// TIA Portal V19 export
FUNCTION "Conv_DT_to_STRING" : String   // FC39, LAD
// stored: Access Published, SetENOAutomatically false
   VAR_INPUT
      Val : DTL;
   END_VAR
   VAR_TEMP
      s_Y : String;
      s_M : String;
      s_D : String;
      s_H : String;
      s_Mi : String;
      s_S : String;
      s_N : String;
      str : String;
   END_VAR
BEGIN

REGION Network 1 (SCL)
   #s_Y := UINT_TO_STRING(#Val.YEAR);
   // Elimina il + a inizio stringa
   #s_Y := MID_STRING(IN := #s_Y, L := LEN(#s_Y) - 1, P := 2);



   #s_M := USINT_TO_STRING(#Val.MONTH);
   // Elimina il + a inizio stringa
   #s_M := MID_STRING(IN := #s_M, L := LEN(#s_M) - 1, P := 2);
   // Aggiunge lo 0 davanti per i mesi da 1 a 9
   IF LEN(#s_M) < 2 THEN
       #s_M := CONCAT(IN1 := '0', IN2 := #s_M);
   END_IF;



   #s_D := USINT_TO_STRING(#Val.DAY);
   // Elimina il + a inizio stringa
   #s_D := MID_STRING(IN := #s_D, L := LEN(#s_D) - 1, P := 2);
   // Aggiunge lo 0 davanti per i giorni da 1 a 9
   IF LEN(#s_D) < 2 THEN
       #s_D := CONCAT(IN1 := '0', IN2 := #s_D);
   END_IF;


   #s_H := USINT_TO_STRING(#Val.HOUR);
   // Elimina il + a inizio stringa
   #s_H := MID_STRING(IN := #s_H, L := LEN(#s_H) - 1, P := 2);
   // Aggiunge lo 0 davanti per le ore da 0 a 9
   IF LEN(#s_H) < 2 THEN
       #s_H := CONCAT(IN1 := '0', IN2 := #s_H);
   END_IF;


   #s_Mi := USINT_TO_STRING(#Val.MINUTE);
   // Elimina il + a inizio stringa
   #s_Mi := MID_STRING(IN := #s_Mi, L := LEN(#s_Mi) - 1, P := 2);
   // Aggiunge lo 0 davanti per i minuti da 0 a 9
   IF LEN(#s_Mi) < 2 THEN
       #s_Mi := CONCAT(IN1 := '0', IN2 := #s_Mi);
   END_IF;



   #s_S := USINT_TO_STRING(#Val.SECOND);
   // Elimina il + a inizio stringa
   #s_S := MID_STRING(IN := #s_S, L := LEN(#s_S) - 1, P := 2);
   // Aggiunge lo 0 davanti per i secondi da 0 a 9
   IF LEN(#s_S) < 2 THEN
       #s_S := CONCAT(IN1 := '0', IN2 := #s_S);
   END_IF;


   #s_N := UDINT_TO_STRING(#Val.NANOSECOND);
   // Elimina il + a inizio stringa
   #s_N := MID_STRING(IN := #s_N, L := LEN(#s_N) - 1, P := 2);
   // Riduci la string a solo 3 caratteri
   #s_N := LEFT(IN := #s_N, L := 3);





   #str := CONCAT(IN1 := #s_Y, IN2 := '-');
   #str := CONCAT(IN1 := #str,IN2:=#s_M);
   #str := CONCAT(IN1 := #str, IN2 := '-');
   #str := CONCAT(IN1 := #str, IN2 := #s_D);
   #str := CONCAT(IN1 := #str, IN2 := ' ');
   #str := CONCAT(IN1 := #str, IN2 := #s_H);
   #str := CONCAT(IN1 := #str, IN2 := ':');
   #str := CONCAT(IN1 := #str, IN2 := #s_Mi);
   #str := CONCAT(IN1 := #str, IN2 := ':');
   #str := CONCAT(IN1 := #str, IN2 := #s_S);
   #str := CONCAT(IN1 := #str, IN2 := '.');
   #str := CONCAT(IN1 := #str, IN2 := #s_N);

   #Conv_DT_to_STRING := #str;
END_REGION
END_FUNCTION
